        "adder2_0"( cin := #c, ain := 5, bin := 8, cout => #c );
        "adder2_1"( cin := #c, ain := 5, bin := 8, cout => #c );
        "adder2_2"( cin := #c, ain := 5, bin := 8, cout => #c );
        "adder2_3"( cin := #c, ain := 5, bin := 8, cout => #c );
        "adder2_4"( cin := #c, ain := 5, bin := 8, cout => #c );
        "adder2_5"( cin := #c, ain := 5, bin := 8, cout => #c );
        "adder2_6"( cin := #c, ain := 5, bin := 8, cout => #c );
        "adder2_7"( cin := #c, ain := 5, bin := 8, cout => #c );
        "adder2_8"( cin := #c, ain := 5, bin := 8, cout => #c );
        "adder2_9"( cin := #c, ain := 5, bin := 8, cout => #c );
        "adder2_10"( cin := #c, ain := 5, bin := 8, cout => #c );
        "adder2_11"( cin := #c, ain := 5, bin := 8, cout => #c );
        "adder2_12"( cin := #c, ain := 5, bin := 8, cout => #c );
        "adder2_13"( cin := #c, ain := 5, bin := 8, cout => #c );
        "adder2_14"( cin := #c, ain := 5, bin := 8, cout => #c );
        "adder2_15"( cin := #c, ain := 5, bin := 8, cout => #c );
        "adder2_16"( cin := #c, ain := 5, bin := 8, cout => #c );
        "adder2_17"( cin := #c, ain := 5, bin := 8, cout => #c );
        "adder2_18"( cin := #c, ain := 5, bin := 8, cout => #c );
        "adder2_19"( cin := #c, ain := 5, bin := 8, cout => #c );
        "adder2_20"( cin := #c, ain := 5, bin := 8, cout => #c );
        "adder2_21"( cin := #c, ain := 5, bin := 8, cout => #c );
        "adder2_22"( cin := #c, ain := 5, bin := 8, cout => #c );
        "adder2_23"( cin := #c, ain := 5, bin := 8, cout => #c );
        "adder2_24"( cin := #c, ain := 5, bin := 8, cout => #c );
        "adder2_25"( cin := #c, ain := 5, bin := 8, cout => #c );
        "adder2_26"( cin := #c, ain := 5, bin := 8, cout => #c );
        "adder2_27"( cin := #c, ain := 5, bin := 8, cout => #c );
        "adder2_28"( cin := #c, ain := 5, bin := 8, cout => #c );
        "adder2_29"( cin := #c, ain := 5, bin := 8, cout => #c );


    END_FOR;
END_ORGANIZATION_BLOCK

